Staubli VAL3: BuildString.pgx

public program BuildString(string x_sInString, string& x_sOutString[], string x_sDelimiter, num& x_nValue[])
  local num l_i
  local num l_n
begin
  // ABSTRACT:
  // This program inserts some real values into a specific string
  //
  // INPUT PARMS:
  //  x_sInString    : Input string into which the real values must be inserted
  //  x_sDelimiter   : Character to be replace by the real value
  //  x_nValue[]     : Real value to be inserted into the input string
  //
  // OUTPUT PARMS:
  //  x_sOutString   : Output string in which the real value ARE inserted
  //
  //Created 21/12/05                              C.CURRIVAND
  //--------------------------------------------------------------
  //
  l_i=0
  x_sOutString=x_sInString
  l_n=find(x_sOutString,x_sDelimiter)
  while (l_i<=size(x_nValue)-1) and (l_n!=-1)
    x_sOutString=replace(x_sOutString,toString("",x_nValue[l_i]),1,l_n)
    l_i=l_i+1
    l_n=find(x_sOutString,x_sDelimiter)
  endWhile
end
